Fanuc KAREL source: kc00041.KL

-- PROVISIONAL review KL for V1013-1; original PC SHA256 d063a8e08af3dca75d4391f9c6a0db42f77345e7a59fd285abd4fb2337a3200c
-- Incomplete behavior may be omitted. Consult companion uncertainty JSON. Do not deploy.
PROGRAM KC00041
%NOLOCKGROUP
BEGIN
  -- UNRESOLVED_PC offsets 5-33; opcodes 27,22,22,22,22,31
  -- UNRESOLVED_PC offsets 38-42; opcodes 7F
END KC00041
